(*

.. <legal notes>

legal notes
=================
| SPDX-FileCopyrightText: © 2025 Oleksandr Tiutyk <trofimich@gmail.com>
| SPDX-License-Identifier: LGPL-3.0-only
| For details check: LGPL-3.0-only_

.. _LGPL-3.0-only: https://www.gnu.org/licenses/lgpl-3.0.en.html

.. </legal notes>

*)

FUNCTION_BLOCK ABSTRACT AutoDisposedObject EXTENDS Object

METHOD FB_init : BOOL
VAR_INPUT
	(* if TRUE, the retain variables are initialized (warm start / cold start)*)
	bInitRetains	: BOOL;
	(* if TRUE, the instance afterwards gets moved into the copy code (online change)*)
	bInCopyCode	: BOOL;
END_VAR
DynamicMemoryManager.RegisterAutoDisposedObject(THIS^);
END_METHOD

END_FUNCTION_BLOCK

(* stored: Version 1.1.0.1
   POU AutoDisposedObject: Id {41c6ec98-296a-4b40-b5dc-94e98a013b84}, SpecialFunc None
   Method FB_init: Id {51ac75a5-4102-427f-b3d7-c1a127754171} *)
